# EPICS autosave request: CARSApp/Db/mono_pid_control_settings.req
# FILE... mono_pid_control_settings.req
file "pid_control_settings.req", P=$(P), PID=$(PID)
$(P)$(PID)EnableReset
